FUNCTION_BLOCK FB_fileReadWrite

VAR_INPUT
	bWrite			: BOOL := FALSE;(* Rising edge starts program execution *)
END_VAR

VAR
	
	sNetId			: T_AmsNetId := '';	(* TwinCAT system network address *)
	sFileRoot		: T_MaxString := 'C:\Users\nbung\Documents\TcXaeShell\CoilWindingMachine\CoilWindingHMI\LOG';
	sFilePath		: T_MaxString := '\';
	sFileName		: T_MaxString := '';(* CSV destination file path and name *) //to do probably should have a way for users to change this
	sCSVLine		: T_MaxString := '';(* Single CSV text line (row, record), we are using string as record buffer (your are able to see created fields) *)
	sCSVField		: T_MaxString := '';(* Single CSV field value (column, record field) *)
	bBusy			: BOOL;
	bError			: BOOL;
	nErrId			: UDINT;
	nRow	 		: UDINT 	:= 0;(* Row number (record) *)
	nColumn			: UDINT 	:= 0;(* Column number (record field) *)
	hFile			: UINT		:= 0;(* File handle of the source file *)
	step			: DWORD 	:= 0;
	stepCheck		: DWORD 	:= 0;
	stepDel: INT;
	fbTimer   : FB_LocalSystemTime := ( bEnable := TRUE, dwCycle := 1 );
	fbFileOpen		: FB_FileOpen;(* Opens file *)
	fbFileClose		: FB_FileClose;(* Closes file *)
	fbFilePuts		: FB_FilePuts;(* Writes one record (line) *)
	fbFileDelete	: FB_FileDelete;(* deletes a file*)
	fbWriter		: FB_CSVMemBufferWriter;(* Helper function block used to create CSV data bytes (single record line) *)
	bDone			: BOOL;
	bCheck          : BOOL;
	bValidPath		: BOOL;
	bDelete			: BOOL;
	database		: ARRAY[0..GVL.MAX_CSV_ROWS, 0..GVL.MAX_CSV_COLUMNS ] OF STRING(GVL.MAX_CSV_FIELD_LENGTH) :=[ 
	'User: ', 'TestUser',
	'Time Started: ', 'N/A', 
	'Time Completed: ', 'N/A',
	'Time Elapsed: ', 'N/A', 
	'Number OF coils: ', 'N/A',
	'Length of coil used: ', 'N/A',
	'User Note: ', 'This is a note from the user. should be last'];
	//system time
	
END_VAR

METHOD checkFile : BOOL
VAR_INPUT
END_VAR
CASE stepCheck OF
	//Waiting for rising edge of writeFile Variable. standby state
	0:
		IF bCheck  THEN
			bDone	:= FALSE;
			bCheck 	:= FALSE;
			bBusy 	:= TRUE;
			bError	:= FALSE;
			nErrId	:= 0;
			hFile	:= 0;
			nRow	:= 0;
			nColumn	:= 0;
			stepCheck 	:= 1;
			
		END_IF
		
	//open file
	1:
		fbFileOpen(bExecute:=FALSE);	
		fbFileOpen(bExecute:=TRUE,
					nmode:=FOPEN_MODEWRITE,
					sPathName:=sFileName,
					sNetId:='',
					tTimeout:=T#5S,); 
		
		stepCheck := 2;
		
		
	//wait untill we are finished opening the text file. 
	2:
		fbFileOpen( bExecute := FALSE, bError => bError, nErrID => nErrID, hFile => hFile );
		IF NOT fbFileOpen.bBusy THEN
			
			IF NOT fbFileOpen.bError THEN
				
				stepCheck := 100;
				bValidPath:=TRUE;
				bDelete :=TRUE;
				
				
			ELSE(* Error: could not create file *)
				stepCheck := 100;
				bValidPath:=FALSE;
				bError:=TRUE;
					
			END_IF
		END_IF

		
	//write single text line.
		10:
		fbFileClose( bExecute := FALSE );
		fbFileClose( sNetId := sNetId, hFile := hFile, bExecute := TRUE );
		stepCheck := 11;
	
	11:(* Wait until close not busy *)
		fbFileClose( bExecute := FALSE, bError => bError, nErrID => nErrID );
		IF ( NOT fbFileClose.bBusy ) THEN
			hFile := 0;
			stepCheck := 100;
		END_IF
	100: (* Error or ready step => cleanup *)
		
		IF ( hFile <> 0 ) THEN
			stepCheck := 10; (* Close the source file *)
		ELSE
			bBusy := FALSE;
			stepCheck := 0;	(* Ready *)
		END_IF
END_CASE
END_METHOD

METHOD CYLIC : BOOL
VAR_INPUT
END_VAR

VAR

t : DATE_AND_TIME ;
END_VAR
fileWrite();
checkFile();
fileDelete();
fbTimer();
END_METHOD

METHOD fileDelete : BOOL
VAR_INPUT
END_VAR

VAR
	
END_VAR
CASE stepDel OF
	//Waiting for rising edge of writeFile Variable. standby state
	0:
		IF bDelete AND NOT bBusy THEN
			bDone	:= FALSE;
			bDelete 	:= FALSE;
			bBusy 	:= TRUE;
			bError	:= FALSE;
			nErrId	:= 0;
			hFile	:= 0;
			
			stepDel 	:= 1;
		END_IF
		
	//open file
	1:
		fbFileDelete(bExecute:=FALSE);
			fbFileDelete(bExecute:=TRUE,	
						sPathName:=sFileName,
						sNetId:='',
						tTimeout:=T#5S,);
		stepDel := 2;
	//wait untill we are finished opening the text file. 
	2:
			fbFileDelete( bExecute := FALSE, bError => bError, nErrID => nErrID );
			IF NOT fbFileDelete.bBusy THEN
			
				IF NOT fbFileDelete.bError THEN
					bDone:=TRUE;
					stepDel :=100;
					
				ELSE(* Error: could not create file *)
				stepDel := 100;
				bValidPath:=FALSE;
				bError:=TRUE;
					
				END_IF
			END_IF
	
	10:
		fbFileClose( bExecute := FALSE );
		fbFileClose( sNetId := sNetId, hFile := hFile, bExecute := TRUE );
		stepDel := 11;
	
	11:(* Wait until close not busy *)
		fbFileClose( bExecute := FALSE, bError => bError, nErrID => nErrID );
		IF ( NOT fbFileClose.bBusy ) THEN
			hFile := 0;
			stepDel := 100;
		END_IF
		
	100: (* Error or ready step => cleanup *)
		bDone:=TRUE;
		IF ( hFile <> 0 ) THEN
			stepDel := 10; (* Close the source file *)
		ELSE
			bBusy := FALSE;
			stepDel := 0;	(* Ready *)
		END_IF
END_CASE
END_METHOD

METHOD fileWrite : BOOL
VAR_INPUT
END_VAR

VAR
 tempString   : STRING;
 newsFilePath : STRING;

 
 
 nDstsize : UDINT;
END_VAR
CASE step OF
	//Waiting for rising edge of writeFile Variable. standby state
	0:
		IF bWrite AND bValidPath THEN
			bDone	:= FALSE;
			bWrite 	:= FALSE;
			bBusy 	:= TRUE;
			bError	:= FALSE;
			nErrId	:= 0;
			hFile	:= 0;
			nRow	:= 0;
			nColumn	:= 0;
			step 	:= 1;
		END_IF
		
	//open file
	1:
		
		tempString := CONCAT('LOG-',WORD_TO_STRING(fbTimer.systemTime.wYear) );
		tempString := CONCAT(tempString, '-');
		tempString := CONCAT(tempString, WORD_TO_STRING(fbTimer.systemTime.wMonth));
		tempString := CONCAT(tempString, '-');
		tempString := CONCAT(tempString, WORD_TO_STRING(fbTimer.systemTime.wDay));
		tempString := CONCAT(tempString, '-');
		tempString := CONCAT(tempString, WORD_TO_STRING(fbTimer.systemTime.wHour));
		tempString := CONCAT(tempString, '-');
		tempString := CONCAT(tempString, WORD_TO_STRING(fbTimer.systemTime.wMinute));
		sFileName := CONCAT('\',tempString);
		findAndReplace(pSrcString:=ADR(sFilePath),pDeleteString:=ADR('/'),pInsertString:=ADR('\'),pDstString:=ADR(newsFilePath),nDstsize:=255);
		sFilePath := CONCAT(sFileRoot,sFilePath);
		sFileName := CONCAT(sFilePath, sFileName);
		
	
		fbFileOpen(bExecute:=FALSE);
		fbFileOpen( sNetId := sNetId,
					sPathName := sFileName, 
					nMode := FOPEN_MODEWRITE OR FOPEN_MODETEXT,(* Open file in TEXT mode! *)
					ePath := PATH_GENERIC,
					bExecute := TRUE );
		step := 2;
	//wait untill we are finished opening the text file. 
	2:
		fbFileOpen( bExecute := FALSE, bError => bError, nErrID => nErrID, hFile => hFile );
		IF NOT fbFileOpen.bBusy THEN
			IF NOT fbFileOpen.bError THEN
				step := 3;
			ELSE(* Error: file not found? *)
				step := 100;
			END_IF
		END_IF
	
	//write single text line.
	3:(* Convert one PLC record to CSV format *)
		sCSVLine := '';
		fbWriter.eCmd := eEnumCmd_First;(* Write first field value *)
		IF nRow <= GVL.MAX_CSV_ROWS THEN

			FOR nColumn := 0 TO GVL.MAX_CSV_COLUMNS BY 1 DO

				sCSVField := STRING_TO_CSVFIELD( database[ nRow, nColumn ], FALSE );(* TODO: Get field value from your application *)

				(* Add new field to the record buffer *)
				fbWriter( 	pBuffer := ADR( sCSVLine ), cbBuffer := SIZEOF( sCSVLine ) - 1, putValue := sCSVField, pValue := 0, cbValue := 0,
							bCRLF := ( nColumn = GVL.MAX_CSV_COLUMNS ) );(* bCRLF == TRUE => Write CRLF after the last field value *)
				IF fbWriter.bOk THEN
					fbWriter.eCmd := eEnumCmd_Next;(* Write next field value *)
				ELSE(* Error *)
					step := 100;
					RETURN;
				END_IF

			END_FOR(* FOR nColumn := 0... *)

			(* FB_FilePuts adds allready CR (carriage return) to the written line.
			We have to replace the $R$L characters with $L character to avoid double CR. *)
			IF RIGHT( sCSVLine, 2 ) = '$R$L' THEN
				sCSVLine := REPLACE( sCSVLine, '$L', 2, LEN( sCSVLine ) - 1 );
			END_IF

			nRow := nRow + 1;(* Increment number of created records (rows) *)
			step := 4;(* Write record to the file *)

		ELSE(* All rows written => Close file *)
			step := 10;
		END_IF

	4:	(* Write single text line *)
	
		fbFilePuts( bExecute := FALSE );
		fbFilePuts( sNetId := sNetId, hFile := hFile, sLine := sCSVLine, bExecute := TRUE );
		step := 5;
	
	//waits for the line of text to finish
	5:
		fbFilePuts( bExecute := FALSE, bError => bError, nErrID => nErrID );
		IF NOT fbFilePuts.bBusy THEN
			IF NOT fbFilePuts.bError THEN
				step := 3;(* Write next record *)
			ELSE(* Error *)
				step := 100;
			END_IF
		END_IF
		
	10:
		fbFileClose( bExecute := FALSE );
		fbFileClose( sNetId := sNetId, hFile := hFile, bExecute := TRUE );
		step := 11;
	
	11:(* Wait until close not busy *)
		fbFileClose( bExecute := FALSE, bError => bError, nErrID => nErrID );
		IF ( NOT fbFileClose.bBusy ) THEN
			hFile := 0;
			step := 100;
		END_IF
		
	100: (* Error or ready step => cleanup *)
		bDone:=TRUE;
		IF ( hFile <> 0 ) THEN
			step := 10; (* Close the source file *)
		ELSE
			bBusy := FALSE;
			step := 0;	(* Ready *)
		END_IF
END_CASE
END_METHOD

METHOD update_database : BOOL
VAR_INPUT
	 
	user : STRING := 'N/A';
	timeStarted : TIME;
	timeCompleted : TIME;
	timeElasped : TIME;
	numOfCoil : INT :=0;
	lengthOCoil : INT :=0;
	userNote : STRING;
END_VAR
database[ 0, 1 ]:=user; //user ID 
database[ 1, 1 ]:=WSTRING_TO_STRING(TIME_TO_WSTRING(timeStarted)); //TO DO this leaves a long in a vauge format. 
database[ 2, 1 ]:=WSTRING_TO_STRING(TIME_TO_WSTRING(timeCompleted));
database[ 3, 1 ]:=WSTRING_TO_STRING(TIME_TO_WSTRING(timeElasped));
database[ 4, 1 ]:=INT_TO_STRING(numOfCoil);
database[ 5, 1 ]:=INT_TO_STRING(lengthOCoil);
database[ 6, 1 ]:=userNote;
END_METHOD

END_FUNCTION_BLOCK

(* stored: Version 1.1.0.1, ProductVersion 3.1.4024.12
   POU FB_fileReadWrite: Id {672718a4-3f7c-4568-983a-5be17c81c63b}, SpecialFunc None
   Method checkFile: Id {10730966-3ca1-4b38-8b1e-b8f40c13e9c6}
   Method CYLIC: Id {022d29b1-9207-44a1-a9b2-dae6b5311cdc}
   Method fileDelete: Id {03752aa4-024a-406f-99e7-ee6c7aa679f0}
   Method fileWrite: Id {7c220b82-3fe5-4faa-8bdb-22d8eb65c323}
   Method update_database: Id {822f2f6a-ee12-4586-a471-9c4d67af88e7} *)
